// TIA Portal V17 export
FUNCTION "FC_VFD_CommFault" : Void   // FC, LAD
{ S7_Optimized_Access := 'TRUE' }
// stored: AutoNumber true
   VAR_TEMP   // added for the SCL form of the ladder/FBD networks
      _w1 : Bool;
      _w2 : Bool;
   END_VAR
BEGIN

REGION Network 1: 变频器通讯故障检测
   // 检测变频器通讯失败/成功的上升沿，置位/复位故障标志；若故障标志保持接通3分钟以上则输出通讯故障报警。
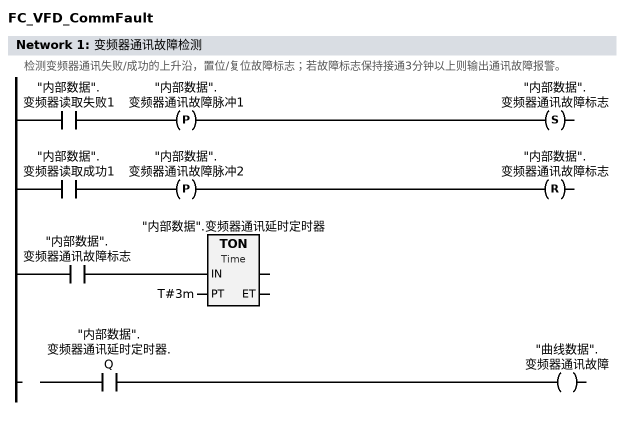
   #_w1 := "内部数据".变频器读取失败1 AND NOT "内部数据".变频器通讯故障脉冲1;   // rising edge
   "内部数据".变频器通讯故障脉冲1 := "内部数据".变频器读取失败1;
   IF #_w1 THEN "内部数据".变频器通讯故障标志 := TRUE; END_IF;
   #_w2 := "内部数据".变频器读取成功1 AND NOT "内部数据".变频器通讯故障脉冲2;   // rising edge
   "内部数据".变频器通讯故障脉冲2 := "内部数据".变频器读取成功1;
   IF #_w2 THEN "内部数据".变频器通讯故障标志 := FALSE; END_IF;
   "内部数据".变频器通讯延时定时器.TON(IN := "内部数据".变频器通讯故障标志, PT := T#3m);
   "曲线数据".变频器通讯故障 := "内部数据".变频器通讯延时定时器.Q;
END_REGION
END_FUNCTION
